(* Logix 5000 project; controller BWFG_Project vendor 1 type 14 code 92 rev 20.13; software revision 20.04; part 2 of 2 *)
(* tags used below, declared in another part *)
   Sequencer : DINT;
   Auto_mode : BOOL;   // Auto Mode Trigger ON/OFF
   Axis_0 : AXIS_SERVO;
   B3 : DINT;   // Hold value for robot Info
   Cabernet_Total : REAL;
   Champagne_Total : REAL;
   Cycle_Complete : ALIAS FOR Robot_Rack:I.Data[0].2;   // Cycle Complete Signal
   Cycle_Start : ALIAS FOR Robot_Rack:O.Data[0].0;   // Cycle start Trigger
   Direction_Mask_Value : DINT;   // the Diresctional Mask for the VFD to change it From Ethernet to Deffalt
   Display_PV : DINT;   // the Display PV screen, used to change the screen
   Drive_Actual_FWD_Speed : REAL;   // Real Speed of the FWD of the driver (in HZ)
   Drive_Actual_REV_Speed : REAL;   // Real Speed of the REV of the driver (in HZ)
   Drive_SPD_Request : REAL;
   ENET_FWD_Speed : DINT;   // the set fwd speed
   ENET_REV_Speed : DINT;   // The set REV speed
   Enet_Speed_HOLD : DINT;
   Entrance_Speed_Select : SINT;
   Event_Driven_Timer : TIMER[14];
   fault_servo_Reset : BOOL;
   FIFO_Bottle_Output : SINT;
   FIFO_Level_Output : SINT;
   FIFO_Location_Output : SINT;
   FIFO_Wine_Output : SINT;
   FWD_REV_Mode : BOOL;   // 0=FWD 1= REV
   Gate_PL : ALIAS FOR Flex_Rack:O.Data[4].4;
   Go_to_Auto_PB : BOOL;   // PV1000+ AUTO SCREEN SELECTED
   GO_to_Display_PB : BOOL;   // PV1000+ DISPALY SCREEN SELECTED
   Go_to_Robot : BOOL;   // PV1000+ ROBOT SCREEN SELECTED
   Goto_Main_PB : BOOL;   // PV1000+ MAIN SCREEN SELECTED
   HMI_indexer : SINT;
   In_Cycle : ALIAS FOR Robot_Rack:I.Data[0].1;
   Level_Percent : REAL;
   Lift_Locate_DOWN_Prox : ALIAS FOR Flex_Rack:I.Data[1].3;   // Lift Locate Down Prox
   Lift_Locate_Prox : ALIAS FOR Flex_Rack:I.Data[1].1;
   Lift_Locate_Raised_Prox : ALIAS FOR Flex_Rack:I.Data[1].2;
   Lift_Locate_UP_Prox : ALIAS FOR Flex_Rack:I.Data[1].2;   // Lift Locate UP Prox
   Location : INT;
   LTU_DOWN_Prox : ALIAS FOR Flex_Rack:I.Data[0].10;   // Lift-transfer-Unit Down Prox
   LTU_Prox : ALIAS FOR Flex_Rack:I.Data[0].9;
   LTU_Raised_Prox : ALIAS FOR Flex_Rack:I.Data[0].11;
   Main_Screen_Button : BOOL;   // PV1000+ MAIN SCREEN SELECTED
   Man_Mode_ON : BOOL;   // PV1000+ MANUAL MODE INDICATOR
   manual_Screen_button : BOOL;   // PV1000+ Manual SCREEN SELECTED
   Merlot_Total : REAL;
   MSG_Display_Num : COUNTER;
   MSG_Timer : TIMER;
   MSG_Timer_2 : TIMER;
   One_Shot : BOOL;
   PF70_Parameter_Value : INT[300];
   PF70_VFD_Control_Mode : SINT;   // VFD Control Mode 0=DIgital / 1 = ENET
   Postion_montior : INT;
   Prestop_Prox : ALIAS FOR Flex_Rack:I.Data[0].8;
   Product_Code : ALIAS FOR Robot_Rack:O.Data[1];
   Pushbutton_Index : BOOL;
   Rest_Seq : BOOL;
   Return_Speed : ALIAS FOR PF70_Parameter_Value[2];   // speed refrence in frequancy
   Robot_Auto_Pass : BOOL;   // allow sequance to work if robot is ready and clear or if bypass is on
   Robot_Bypass : BOOL;   // Skips Robot in sequance if ON
   Robot_Bypass_PB : BOOL;   // Robot Baypass button allowing robot to be skiped
   Robot_Clear : ALIAS FOR Robot_Rack:I.Data[0].0;   // checks if robot is clear of orignal program and is ready to start
   Robot_Message : SINT;
   RPM : REAL;
   Seq_Step : DINT[14];
   Sequencer_Output : DINT;
   Servo_ACC : INT;
   Servo_Control : MOTION_INSTRUCTION[10];
   Servo_Dec : INT;
   Servo_Postion : REAL;
   Servo_Speed : INT;
   Speed_Select_Conferm : BOOL;
   SQO_Control : CONTROL;
   SQO_Mask : DINT;
   Status_Message : ALIAS FOR Robot_Rack:I.Data[1];
   Transfer_Prestop_Prox : ALIAS FOR Flex_Rack:I.Data[1].8;
   Variables : SINT[12];
   VFD_FWD_Hold : SINT;
   VFD_Message : MESSAGE;
   VFD_Message_2 : MESSAGE;
   VFD_REV_Hold : SINT;
   Wine_Total_1 : BOOL;
   Wine_Total_2 : BOOL;
   Wine_Total_3 : BOOL;
(* MainProgram, continued *)

ROUTINE Robot   (* ladder *)
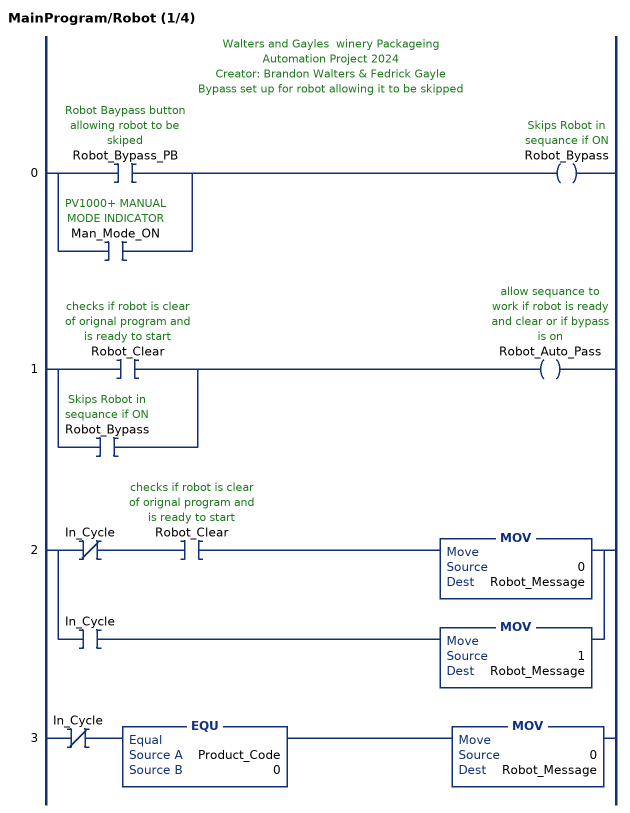
   // Walters and Gayles  winery Packageing
   // Automation Project 2024
   // Creator: Brandon Walters & Fedrick Gayle
   // Bypass set up for robot allowing it to be skipped
   0: [XIC(Robot_Bypass_PB) ,XIC(Man_Mode_ON) ]OTE(Robot_Bypass);
   1: [XIC(Robot_Clear) ,XIC(Robot_Bypass) ]OTE(Robot_Auto_Pass);
   2: [XIO(In_Cycle) XIC(Robot_Clear) MOV(0,Robot_Message) ,XIC(In_Cycle) MOV(1,Robot_Message) ];
   3: XIO(In_Cycle)EQU(Product_Code,0)MOV(0,Robot_Message);
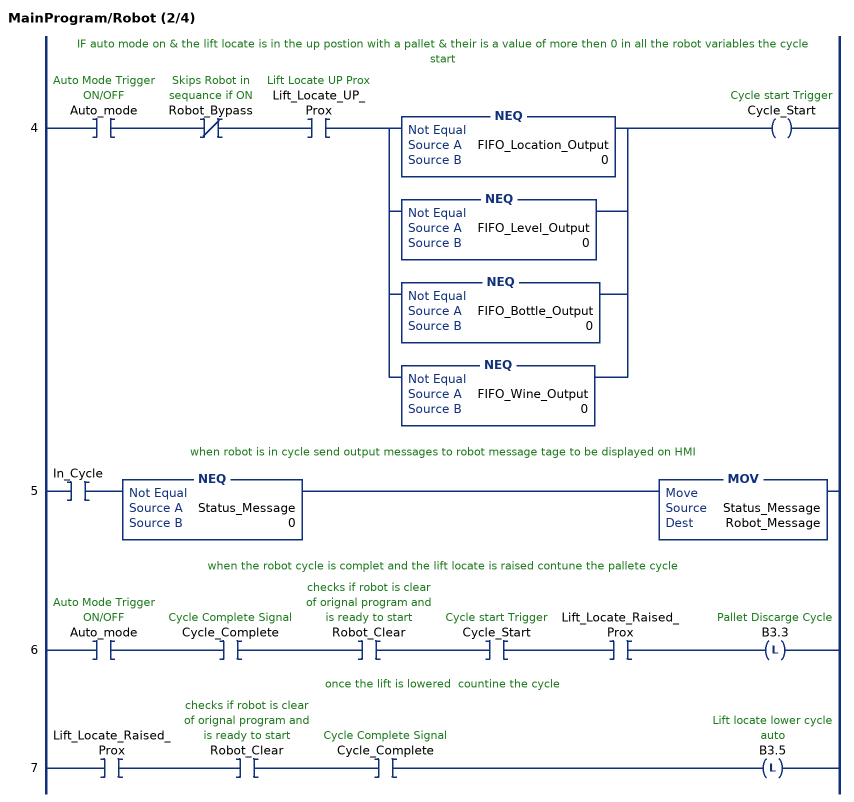
   // IF auto mode on & the lift locate is in the up postion with a pallet & their is a value of more then 0 in all the robot variables the cycle start
   4: XIC(Auto_mode)XIO(Robot_Bypass)XIC(Lift_Locate_UP_Prox)[NEQ(FIFO_Location_Output,0) ,NEQ(FIFO_Level_Output,0) ,NEQ(FIFO_Bottle_Output,0) ,NEQ(FIFO_Wine_Output,0) ]OTE(Cycle_Start);
   // when robot is in cycle send output messages to robot message tage to be displayed on HMI
   5: XIC(In_Cycle)NEQ(Status_Message,0)MOV(Status_Message,Robot_Message);
   // when the robot cycle is complet and the lift locate is raised contune the pallete cycle
   6: XIC(Auto_mode)XIC(Cycle_Complete)XIC(Robot_Clear)XIC(Cycle_Start)XIC(Lift_Locate_Raised_Prox)OTL(B3.3);
   // once the lift is lowered  countine the cycle
   7: XIC(Lift_Locate_Raised_Prox)XIC(Robot_Clear)XIC(Cycle_Complete)OTL(B3.5);
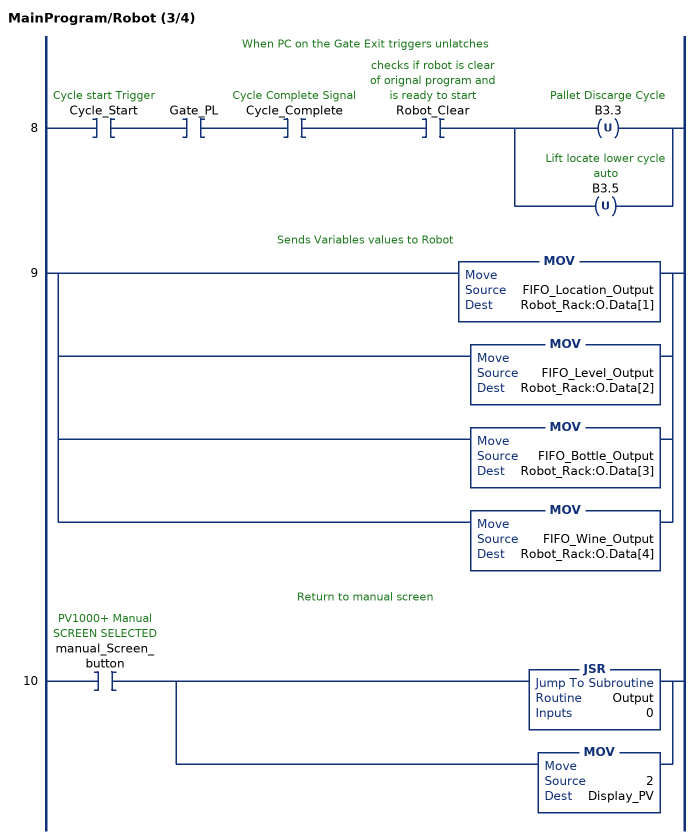
   // When PC on the Gate Exit triggers unlatches
   8: XIC(Cycle_Start)XIC(Gate_PL)XIC(Cycle_Complete)XIC(Robot_Clear)[OTU(B3.3) ,OTU(B3.5) ];
   // Sends Variables values to Robot
   9: [MOV(FIFO_Location_Output,Robot_Rack:O.Data[1]) ,MOV(FIFO_Level_Output,Robot_Rack:O.Data[2]) ,MOV(FIFO_Bottle_Output,Robot_Rack:O.Data[3]) ,MOV(FIFO_Wine_Output,Robot_Rack:O.Data[4]) ];
   // Return to manual screen
   10: XIC(manual_Screen_button)[JSR(Output,0) ,MOV(2,Display_PV) ];
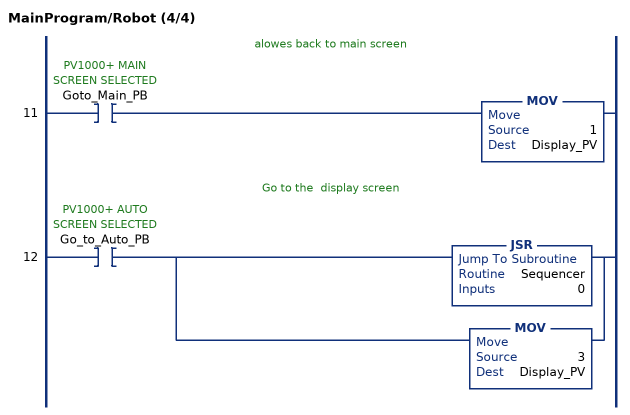
   // alowes back to main screen
   11: XIC(Goto_Main_PB)MOV(1,Display_PV);
   // Go to the  display screen
   12: XIC(Go_to_Auto_PB)[JSR(Sequencer,0) ,MOV(3,Display_PV) ];
END_ROUTINE

ROUTINE Sequencer   (* ladder *)
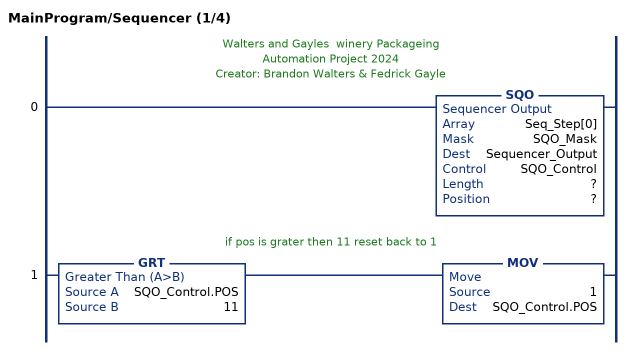
   // Walters and Gayles  winery Packageing
   // Automation Project 2024
   // Creator: Brandon Walters & Fedrick Gayle
   0: SQO(Seq_Step[0],SQO_Mask,Sequencer_Output,SQO_Control,?,?);
   // if pos is grater then 11 reset back to 1
   1: GRT(SQO_Control.POS,11)MOV(1,SQO_Control.POS);
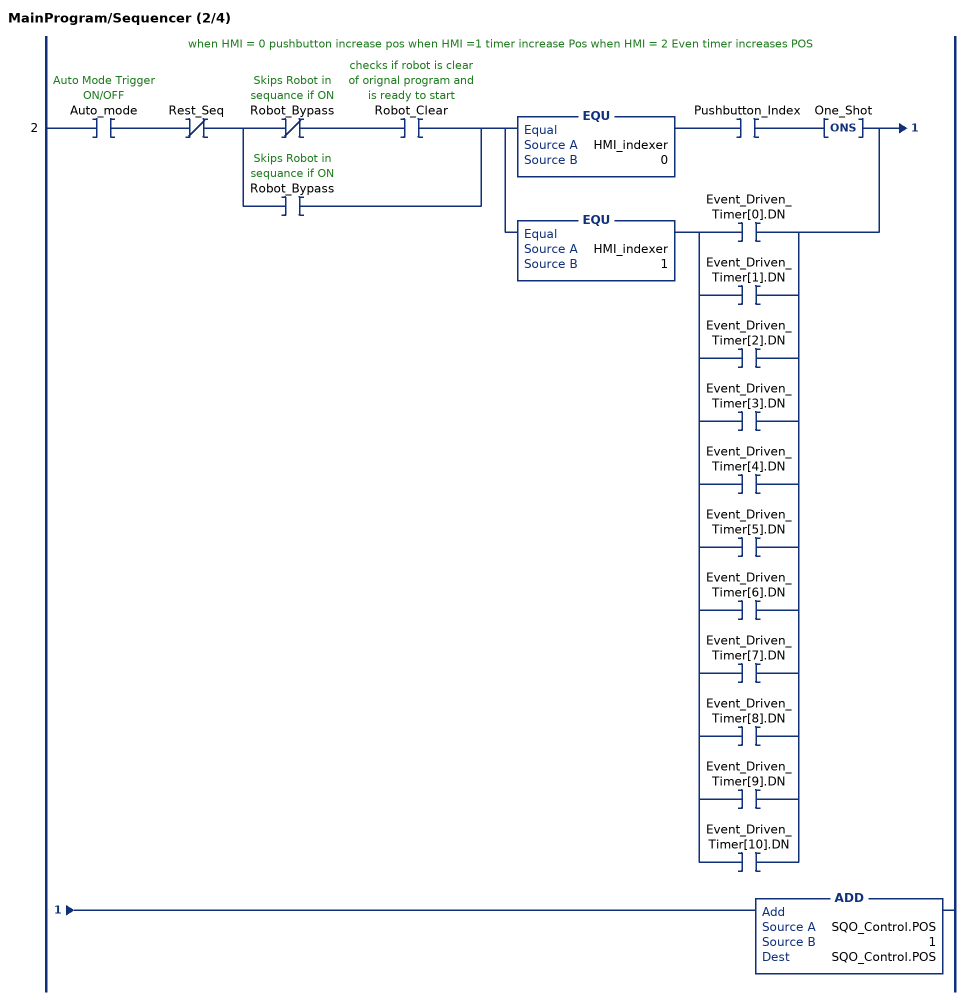
   // when HMI = 0 pushbutton increase pos when HMI =1 timer increase Pos when HMI = 2 Even timer increases POS
   2: XIC(Auto_mode)XIO(Rest_Seq)[XIO(Robot_Bypass) XIC(Robot_Clear) ,XIC(Robot_Bypass) ][EQU(HMI_indexer,0) XIC(Pushbutton_Index) ONS(One_Shot) ,EQU(HMI_indexer,1) [XIC(Event_Driven_Timer[0].DN) ,XIC(Event_Driven_Timer[1].DN) ,XIC(Event_Driven_Timer[2].DN) ,XIC(Event_Driven_Timer[3].DN) ,XIC(Event_Driven_Timer[4].DN) ,XIC(Event_Driven_Timer[5].DN) ,XIC(Event_Driven_Timer[6].DN) ,XIC(Event_Driven_Timer[7].DN) ,XIC(Event_Driven_Timer[8].DN) ,XIC(Event_Driven_Timer[9].DN) ,XIC(Event_Driven_Timer[10].DN) ] ]ADD(SQO_Control.POS,1,SQO_Control.POS);
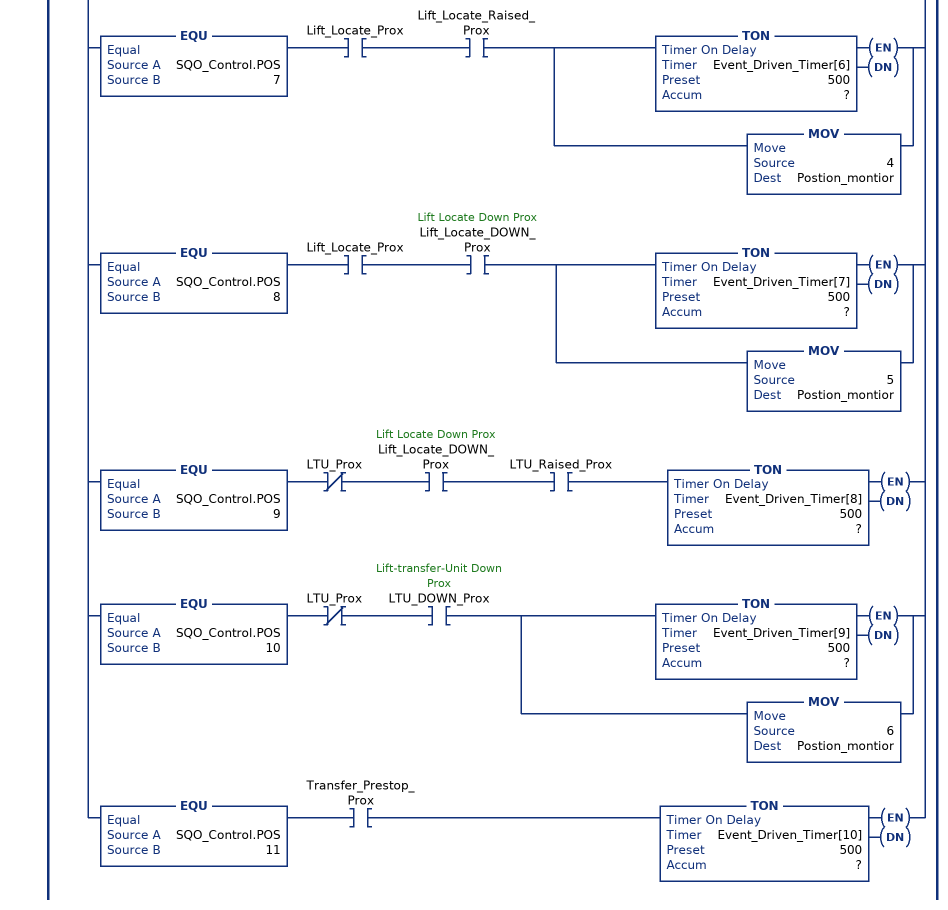
   // envent triggering based on location
   3: XIC(Auto_mode)XIO(Rest_Seq)EQU(HMI_indexer,1)[EQU(SQO_Control.POS,1) XIC(Prestop_Prox) [TON(Event_Driven_Timer[0],?,?) ,MOV(1,Postion_montior) ] ,EQU(SQO_Control.POS,2) XIC(Prestop_Prox) TON(Event_Driven_Timer[1],?,?) ,EQU(SQO_Control.POS,3) XIO(LTU_Prox) [TON(Event_Driven_Timer[2],?,?) ,MOV(2,Postion_montior) ] ,EQU(SQO_Control.POS,4) XIO(LTU_Prox) TON(Event_Driven_Timer[3],?,?) ,EQU(SQO_Control.POS,5) XIO(LTU_Prox) XIC(LTU_Raised_Prox) [TON(Event_Driven_Timer[4],?,?) ,MOV(3,Postion_montior) ] ,EQU(SQO_Control.POS,6) XIC(Lift_Locate_Prox) TON(Event_Driven_Timer[5],?,?) ,EQU(SQO_Control.POS,7) XIC(Lift_Locate_Prox) XIC(Lift_Locate_Raised_Prox) [TON(Event_Driven_Timer[6],?,?) ,MOV(4,Postion_montior) ] ,EQU(SQO_Control.POS,8) XIC(Lift_Locate_Prox) XIC(Lift_Locate_DOWN_Prox) [TON(Event_Driven_Timer[7],?,?) ,MOV(5,Postion_montior) ] ,EQU(SQO_Control.POS,9) XIO(LTU_Prox) XIC(Lift_Locate_DOWN_Prox) XIC(LTU_Raised_Prox) TON(Event_Driven_Timer[8],?,?) ,EQU(SQO_Control.POS,10) XIO(LTU_Prox) XIC(LTU_DOWN_Prox) [TON(Event_Driven_Timer[9],?,?) ,MOV(6,Postion_montior) ] ,EQU(SQO_Control.POS,11) XIC(Transfer_Prestop_Prox) TON(Event_Driven_Timer[10],?,?) ];
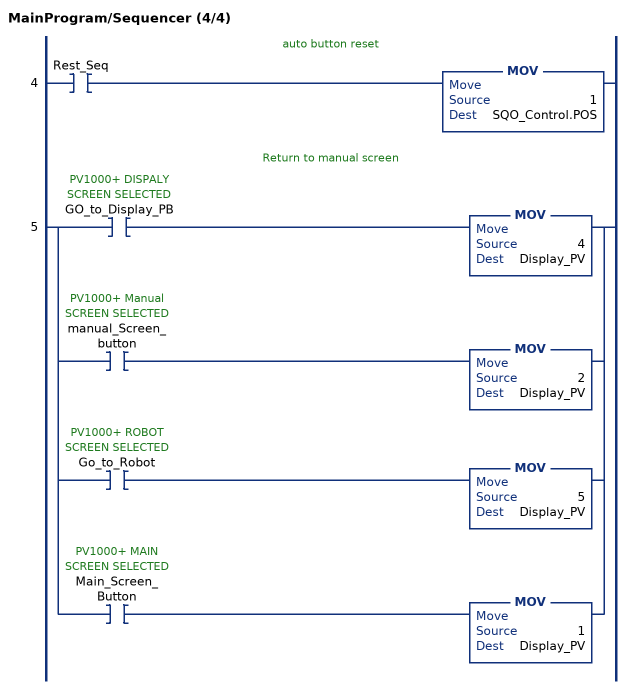
   // auto button reset
   4: XIC(Rest_Seq)MOV(1,SQO_Control.POS);
   // Return to manual screen
   5: [XIC(GO_to_Display_PB) MOV(4,Display_PV) ,XIC(manual_Screen_button) MOV(2,Display_PV) ,XIC(Go_to_Robot) MOV(5,Display_PV) ,XIC(Main_Screen_Button) MOV(1,Display_PV) ];
END_ROUTINE

ROUTINE Servo   (* ladder *)
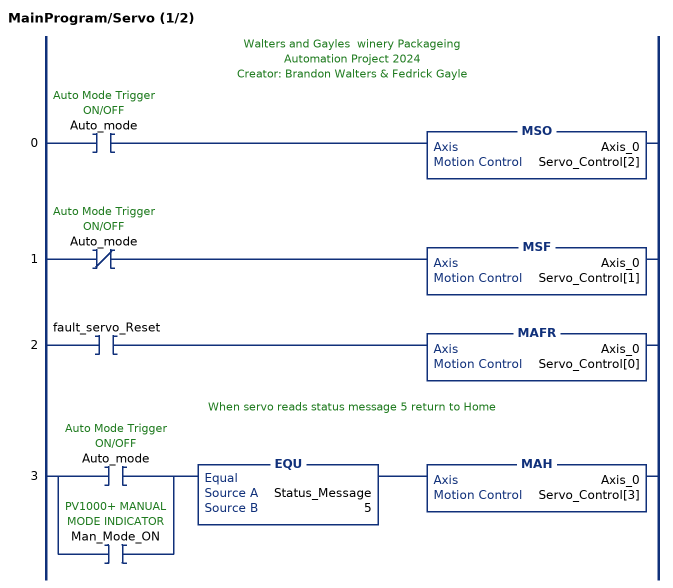
   // Walters and Gayles  winery Packageing
   // Automation Project 2024
   // Creator: Brandon Walters & Fedrick Gayle
   0: XIC(Auto_mode)MSO(Axis_0,Servo_Control[2]);
   1: XIO(Auto_mode)MSF(Axis_0,Servo_Control[1]);
   2: XIC(fault_servo_Reset)MAFR(Axis_0,Servo_Control[0]);
   // When servo reads status message 5 return to Home
   3: [XIC(Auto_mode) ,XIC(Man_Mode_ON) ]EQU(Status_Message,5)MAH(Axis_0,Servo_Control[3]);
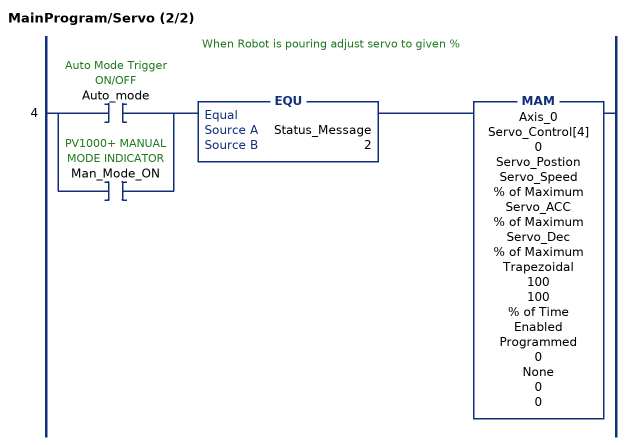
   // When Robot is pouring adjust servo to given %
   4: [XIC(Auto_mode) ,XIC(Man_Mode_ON) ]EQU(Status_Message,2)MAM(Axis_0,Servo_Control[4],0,Servo_Postion,Servo_Speed,% of Maximum,Servo_ACC,% of Maximum,Servo_Dec,% of Maximum,Trapezoidal,100,100,% of Time,Enabled,Programmed,0,None,0,0);
END_ROUTINE

ROUTINE speed_sel_calc   (* function block diagram *)
   SHEET 1
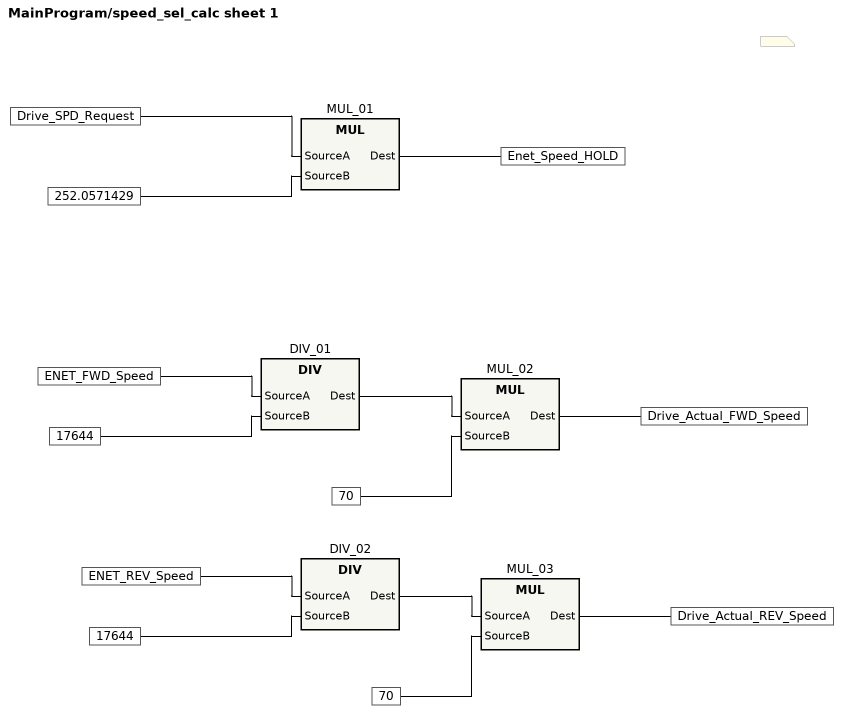
   DIV_01 : DIV(SourceA := ENET_FWD_Speed, SourceB := 17644);
   MUL_01 : MUL(SourceA := Drive_SPD_Request, SourceB := 252.0571429);
   DIV_02 : DIV(SourceA := ENET_REV_Speed, SourceB := 17644);
   MUL_02 : MUL(SourceA := DIV_01.Dest, SourceB := 70);
   MUL_03 : MUL(SourceA := DIV_02.Dest, SourceB := 70);
   Enet_Speed_HOLD := MUL_01.Dest;
   Drive_Actual_FWD_Speed := MUL_02.Dest;
   Drive_Actual_REV_Speed := MUL_03.Dest;
END_ROUTINE

ROUTINE Speed_Select   (* ladder *)
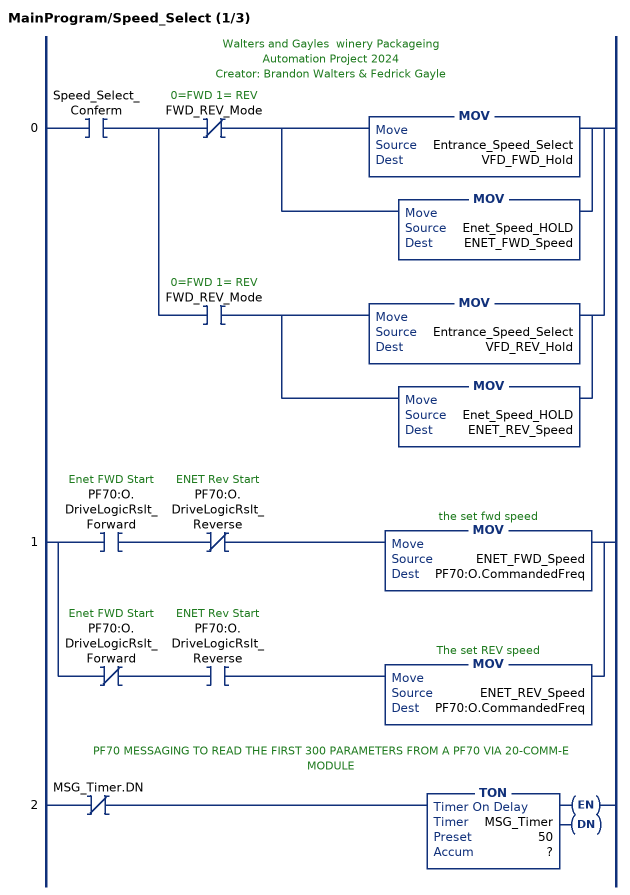
   // Walters and Gayles  winery Packageing
   // Automation Project 2024
   // Creator: Brandon Walters & Fedrick Gayle
   0: XIC(Speed_Select_Conferm)[XIO(FWD_REV_Mode) [MOV(Entrance_Speed_Select,VFD_FWD_Hold) ,MOV(Enet_Speed_HOLD,ENET_FWD_Speed) ] ,XIC(FWD_REV_Mode) [MOV(Entrance_Speed_Select,VFD_REV_Hold) ,MOV(Enet_Speed_HOLD,ENET_REV_Speed) ] ];
   1: [XIC(PF70:O.DriveLogicRslt_Forward) XIO(PF70:O.DriveLogicRslt_Reverse) MOV(ENET_FWD_Speed,PF70:O.CommandedFreq) ,XIO(PF70:O.DriveLogicRslt_Forward) XIC(PF70:O.DriveLogicRslt_Reverse) MOV(ENET_REV_Speed,PF70:O.CommandedFreq) ];
   // PF70 MESSAGING TO READ THE FIRST 300 PARAMETERS FROM A PF70 VIA 20-COMM-E MODULE
   2: XIO(MSG_Timer.DN)TON(MSG_Timer,?,?);
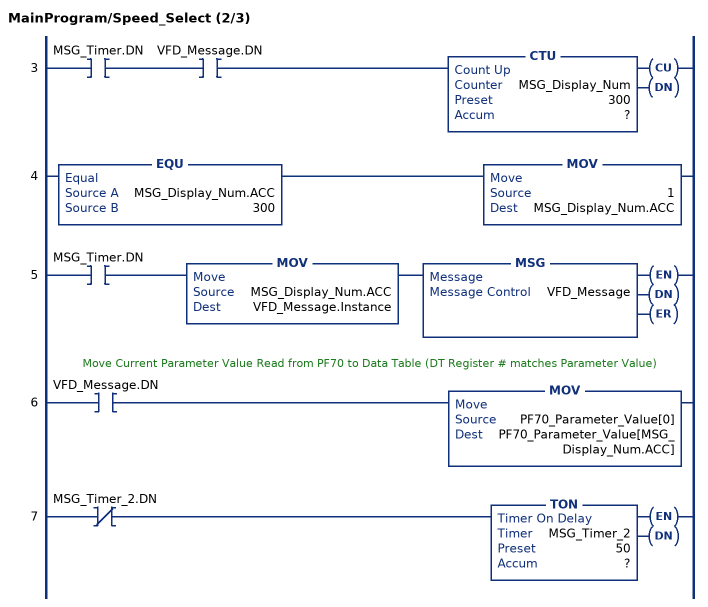
   3: XIC(MSG_Timer.DN)XIC(VFD_Message.DN)CTU(MSG_Display_Num,?,?);
   4: EQU(MSG_Display_Num.ACC,300)MOV(1,MSG_Display_Num.ACC);
   5: XIC(MSG_Timer.DN)MOV(MSG_Display_Num.ACC,VFD_Message.Instance)MSG(VFD_Message);
   // Move Current Parameter Value Read from PF70 to Data Table (DT Register # matches Parameter Value)
   6: XIC(VFD_Message.DN)MOV(PF70_Parameter_Value[0],PF70_Parameter_Value[MSG_Display_Num.ACC]);
   7: XIO(MSG_Timer_2.DN)TON(MSG_Timer_2,?,?);
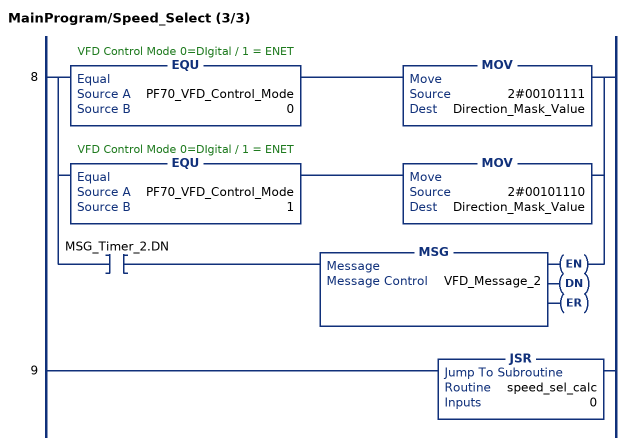
   8: [[EQU(PF70_VFD_Control_Mode,0) MOV(2#00101111,Direction_Mask_Value) ,EQU(PF70_VFD_Control_Mode,1) MOV(2#00101110,Direction_Mask_Value) ] ,XIC(MSG_Timer_2.DN) MSG(VFD_Message_2) ];
   9: JSR(speed_sel_calc,0);
END_ROUTINE

ROUTINE Tank_info   (* structured text *)
   //Walters and Gayles  winery Packageing
   //Automation Project 2024
   //Creator: Brandon Walters & Fedrick Gayle
   Level_Percent:= FIFO_Level_Output * 0.1;
   If Wine_Total_1 Then //If robot in pour and wine 1 was selected reduce total amount by % given
   Merlot_Total:= Merlot_Total - (Level_Percent); // total amount of wine - fill percent
   ELSIF Wine_Total_2 Then
   Champagne_Total:= Champagne_Total - (Level_Percent);// total amount of wine - fill percent
   ELSIF Wine_Total_3 Then
   Cabernet_Total:= Cabernet_Total - (Level_Percent);// total amount of wine - fill percent
   END_IF;
   
   
   RPM:= (120*((Return_Speed/17644)*70)/4)/60;// RPM calculation for speed
   Servo_Postion:= 7*(FIFO_Level_Output/100);// servo calculation for adjusting postion based on given %
   
END_ROUTINE
END_PROGRAM
